FUNCTION_BLOCK Mover IMPLEMENTS I_Mover
VAR
	{attribute 'hide'}
	_Parameters : ParameterSet;
	{attribute 'hide'}
	_Status		: ParameterSet;
	{attribute 'hide'}
	_PointerExample : BOOL;
	testTask	: InterfaceTaskExample(_Parameters, _Status);
	pointerTask : PointerTaskExample(THIS^);
END_VAR

METHOD CyclicLogic
VAR_INPUT
END_VAR
IF _PointerExample THEN
	pointerTask.CyclicLogic();
	RETURN;
END_IF

testTask.CyclicLogic();
END_METHOD

{attribute 'monitoring':='call'}
PROPERTY Parameters : I_ParameterPosition
GET
Parameters := _Parameters;
END_GET
SET
END_SET
END_PROPERTY

{attribute 'monitoring':='call'}
PROPERTY PointerExample : BOOL
GET
PointerExample := _PointerExample;
END_GET
SET
_PointerExample := PointerExample;
END_SET
END_PROPERTY

{attribute 'monitoring':='call'}
PROPERTY Status : I_ParameterPositionGetter
GET
Status := _Status;
END_GET
END_PROPERTY

END_FUNCTION_BLOCK

(* stored: Version 1.1.0.1
   POU Mover: Id {d30ab331-ed7a-4c35-aedc-6533f8ef6904}, SpecialFunc None
   Method CyclicLogic: Id {c730d094-6adb-42c6-9852-80118348f8f4}
   Property Parameters: Id {64adcffc-21ec-43d1-8a59-70cb5447c9be}
   Get Get: Id {3fe304cc-925e-4aae-90c4-7d1e4770e87f}
   Set Set: Id {b13ed811-dfa1-4f62-b719-a5488a84c30e}
   Property PointerExample: Id {632eaa34-f068-460e-81ad-c49321734460}
   Get Get: Id {fd642448-fc89-4cf1-b371-78ed23962109}
   Set Set: Id {19f2b6ca-85c5-4aed-96f0-6aaf7df0dbbd}
   Property Status: Id {6b45aeb4-f49b-44f5-8f31-961f135833f7}
   Get Get: Id {2cdb6f3e-c43a-42c0-9ee1-395514dc5d17} *)
